TYPE st_router_data :
STRUCT
	Device 		: 	st_Device;
	GPS			:	st_GPS;
	Mobile		:	st_mobile;
	e_SMSStatus : 	eSMSStatus;
	Events		:	st_TeltonikaEvents;
END_STRUCT
END_TYPE

(* stored: Version 1.1.0.1, ProductVersion 3.1.4024.12
   DUT st_router_data: Id {acfc0de7-5474-49bd-b092-b098fdfbac71} *)
